FUNCTION_BLOCK NCTController EXTENDS CyclicBase
VAR
	_MyInterface: Tc3_XTS_Utility.I_TcIoXtsNctBaseUnitInterface;
END_VAR


//_MyInterface := _MyXpu.NctControllerTcIo().BaseUnitInterfaceTcIo(1);

PROPERTY MyXtsIoInterface : I_TcIoXtsNctBaseUnitInterface
GET
MyXtsIoInterface := _MyInterface;
END_GET
SET
_MyInterface := MyXtsIoInterface;
END_SET
END_PROPERTY

END_FUNCTION_BLOCK

(* stored: Version 1.1.0.1
   POU NCTController: Id {69fac2e2-98e3-4a73-9148-7a9f4979e9be}, SpecialFunc None
   Property MyXtsIoInterface: Id {6c7dd504-29ec-421f-85ee-ffbaf90d2e30}
   Get Get: Id {f25cbf22-78df-4612-a07b-0c830e2b4a03}
   Set Set: Id {f3bbd975-6c48-412c-bf19-c0d38fee92f8} *)
